// TIA Portal project "Anwenderseite" (V16)

(* hardware
DEVICE "S7-1200-Station_1"  S7-1200 Station
   slot 0: "Baugruppenträger_0"  S7-1200 Rack  Rack  V1.0
   slot 1: "PLC_1"  CPU 1214C DC/DC/DC  6ES7 214-1AG40-0XB0  V4.4
*)

// ===== PLC "PLC_1"  CPU 1214C DC/DC/DC =====

VAR_GLOBAL   // PLC tag table "Standard-Variablentabelle"
   "START" AT %M0.0 : Bool;
   "STOP" AT %M0.1 : Bool;
   "MOTOR" AT %Q0.0 : Bool;
   "ERR" AT %MW2 : Int;
END_VAR

ORGANIZATION_BLOCK "Main"   // OB1, FBD, ProgramCycle
TITLE = "Main Program Sweep (Cycle)"
{ S7_Optimized_Access := 'TRUE' }
VERSION : 0.1
   VAR_INPUT
      Initial_Call : Bool;   // Initial call of this OB
      Remanence : Bool;   // =True, if remanent data are available
   END_VAR
BEGIN

REGION Network 1
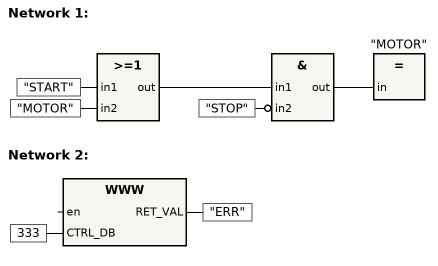
   "MOTOR" := ("START" OR "MOTOR") AND NOT "STOP";
END_REGION

REGION Network 2
   "ERR" := WWW(CTRL_DB := 333);
END_REGION
END_ORGANIZATION_BLOCK